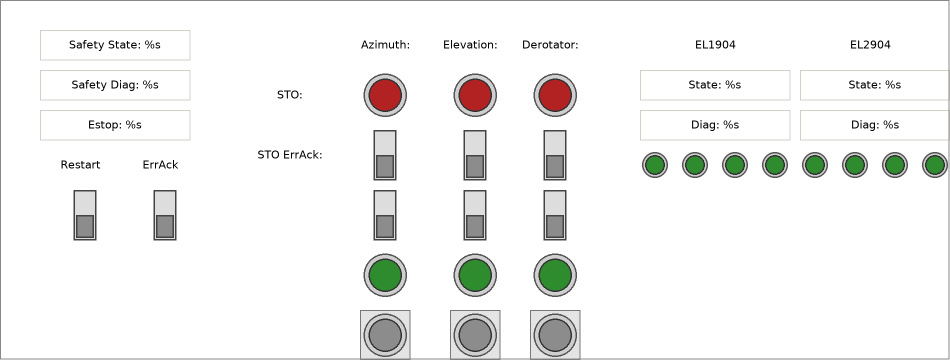
VISUALIZATION Safety  // 950x360
    Label (340,30 91x30), "Azimuth:"
    Lamp1 (360,70 50x50), variable: GVL_Telescope.Azimuth_sto, style: Lamp-Lamp1-Red
    Label (430,30 81x30), "Elevation:"
    Lamp1 (450,70 50x50), variable: GVL_Telescope.Elevation_sto, style: Lamp-Lamp1-Red
    Label (510,30 81x30), "Derotator:"
    Lamp1 (530,70 50x50), variable: GVL_Telescope.Derotator_sto, style: Lamp-Lamp1-Red
    Label (240,80 100x30), "STO:"
    Lamp1 (360,250 50x50), variable: AzimuthElevationControl.ready, style: Lamp-Lamp1-Green
    Lamp1 (450,250 50x50), variable: ElevationControl.Ready, style: Lamp-Lamp1-Green
    Lamp1 (530,250 50x50), style: Lamp-Lamp1-Green
    PushSwitch (360,310 50x50), variable: AzimuthElevationControl.Reset, behaviour: TAP, style: Switch-PushSwitch-Gray
    PushSwitch (450,310 50x50), variable: ElevationControl.reset, behaviour: TAP, style: Switch-PushSwitch-Gray
    PushSwitch (530,310 50x50), behaviour: TAP, style: Switch-PushSwitch-Gray
    DipSwitch (360,190 50x50), variable: AzimuthElevationControl.Enable, behaviour: TOGGLE, style: Switch-DipSwitch-Gray
    DipSwitch (450,190 50x50), variable: ElevationControl.enable, behaviour: TOGGLE, style: Switch-DipSwitch-Gray
    DipSwitch (530,190 50x50), variable: DerotatorControl.enable, behaviour: TOGGLE, style: Switch-DipSwitch-Gray
    DipSwitch (60,190 50x50), variable: GVL_Safety.Restart, behaviour: TOGGLE, style: Switch-DipSwitch-Gray
    DipSwitch (530,130 50x50), variable: GVL_Safety.Reset_STO_Derotator, behaviour: TOGGLE, style: Switch-DipSwitch-Gray
    DipSwitch (360,130 50x50), variable: GVL_Safety.Reset_STO_Azimuth, behaviour: TOGGLE, style: Switch-DipSwitch-Gray
    DipSwitch (450,130 50x50), variable: GVL_Safety.Reset_STO_Elevation, behaviour: TOGGLE, style: Switch-DipSwitch-Gray
    Label (240,140 100x30), "STO ErrAck:"
    Label (40,150 81x30), "Restart"
    DipSwitch (140,190 50x50), variable: GVL_Safety.ErrAck, behaviour: TOGGLE, style: Switch-DipSwitch-Gray
    Label (120,150 81x30), "ErrAck"
    Textfield (40,30 150x30), "Safety State: %s", text variable: SafetyHandling.fbInfoEStop1.sState, input disabled if: TRUE
    Textfield (40,110 150x30), "Estop: %s", text variable: SafetyHandling.fbInfoEStop1.sState, input disabled if: TRUE
    Textfield (40,70 150x30), "Safety Diag: %s", text variable: SafetyHandling.fbInfoEStop1.sDiag, input disabled if: TRUE
    Label (670,30 91x30), "EL1904"
    Label (830,30 81x30), "EL2904"
    Textfield (640,70 150x30), "State: %s", text variable: SafetyHandling.fbInfoSafetyIn.sState, input disabled if: TRUE
    Textfield (640,110 150x30), "Diag: %s", text variable: SafetyHandling.fbInfoSafetyIn.sDiag, input disabled if: TRUE
    Textfield (800,70 150x30), "State: %s", text variable: SafetyHandling.fbInfoSafetyOut.sState, input disabled if: TRUE
    Textfield (800,110 150x30), "Diag: %s", text variable: SafetyHandling.fbInfoSafetyOut.sDiag, input disabled if: TRUE
    Lamp1 (640,150 30x30), variable: SafetyHandling.bSafetyInCh1, style: Lamp-Lamp1-Green
    Lamp1 (680,150 30x30), variable: SafetyHandling.bSafetyInCh2, style: Lamp-Lamp1-Green
    Lamp1 (720,150 30x30), variable: SafetyHandling.bSafetyInCh3, style: Lamp-Lamp1-Green
    Lamp1 (760,150 30x30), variable: SafetyHandling.bSafetyInCh4, style: Lamp-Lamp1-Green
    Lamp1 (800,150 30x30), variable: SafetyHandling.bSafetyInCh1, style: Lamp-Lamp1-Green
    Lamp1 (840,150 30x30), variable: SafetyHandling.bSafetyInCh2, style: Lamp-Lamp1-Green
    Lamp1 (880,150 30x30), variable: SafetyHandling.bSafetyInCh3, style: Lamp-Lamp1-Green
    Lamp1 (920,150 30x30), variable: SafetyHandling.bSafetyInCh4, style: Lamp-Lamp1-Green
END_VISUALIZATION

(* stored: Version 1.1.0.1, ProductVersion 3.1.4024.12
   Visu Safety: Id {2c72abb1-52b7-4434-8d69-25eedaf9331f} *)
